// TIA Portal V17 export
// export: Created 2023-11-12T16:12:26.0840163Z, ExportSetting WithDefaults, DisplayName Totally Integrated Automation Portal, DisplayVersion V17, DisplayName TIA Portal Openness, DisplayVersion V17, DisplayName TIA Portal Version Control Interface, DisplayVersion V17, DisplayName SINAMICS Startdrive Advanced, DisplayVersion V17 Update2, DisplayName SINAMICS Startdrive G130, G150, S120, S150, SINAMICS MV, S210, DisplayVersion V17 Update2, DisplayName SINAMICS Startdrive G110M, G120, G120C, G120D, G120P, G115D, DisplayVersion V17 Update2, DisplayName STEP 7 Professional, DisplayVersion V17, DisplayName STEP 7 Safety, DisplayVersion V17, DisplayName WinCC Advanced / Unified PC, DisplayVersion V17
ORGANIZATION_BLOCK "Main"   // OB1, LAD, ProgramCycle
TITLE = "Main Program Sweep (Cycle)"
{ S7_Optimized_Access := 'TRUE' }
VERSION : 0.1
// stored: AutoNumber true, IsIECCheckEnabled false, SetENOAutomatically false
   VAR_INPUT
      Initial_Call : Bool;   // Initial call of this OB
      Remanence : Bool;   // =True, if remanent data are available
   END_VAR
   VAR_TEMP
      SOME_BOOLEAN : Bool;
   END_VAR
BEGIN

REGION Network 1
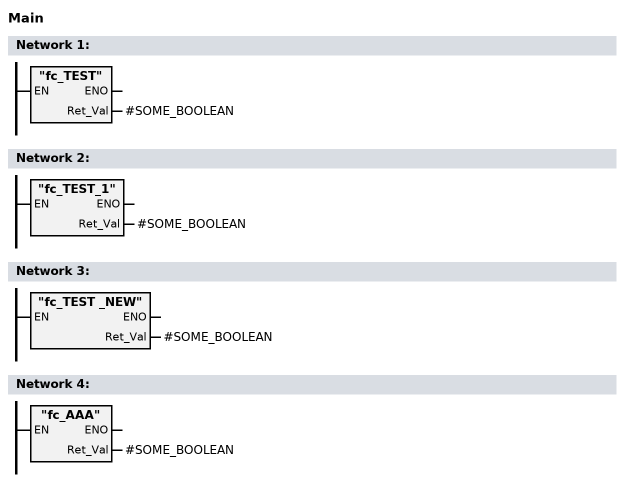
   RUNG wire#powerrail
      "fc_TEST"(Ret_Val => #SOME_BOOLEAN)
   END_RUNG
   // the same network as SCL:
   #SOME_BOOLEAN := "fc_TEST"();
END_REGION

REGION Network 2
   RUNG wire#powerrail
      "fc_TEST_1"(Ret_Val => #SOME_BOOLEAN)
   END_RUNG
   // the same network as SCL:
   #SOME_BOOLEAN := "fc_TEST_1"();
END_REGION

REGION Network 3
   RUNG wire#powerrail
      "fc_TEST _NEW"(Ret_Val => #SOME_BOOLEAN)
   END_RUNG
   // the same network as SCL:
   #SOME_BOOLEAN := "fc_TEST _NEW"();
END_REGION

REGION Network 4
   RUNG wire#powerrail
      "fc_AAA"(Ret_Val => #SOME_BOOLEAN)
   END_RUNG
   // the same network as SCL:
   #SOME_BOOLEAN := "fc_AAA"();
END_REGION
END_ORGANIZATION_BLOCK
